	//
	IF _CmdParams[2] = _LiteralString THEN
		// file1.cnc XYZ H +0250.00 +0000.00 +0500.00 +0000.00 +0045.00 +0180.00
		stCommand.StartPos.dX:=STRING_TO_LREAL(_CmdParams[3]);
		stCommand.StartPos.dY:=STRING_TO_LREAL(_CmdParams[4]);
		stCommand.StartPos.dZ:=STRING_TO_LREAL(_CmdParams[5]);
		stCommand.StartPos.dA:=STRING_TO_LREAL(_CmdParams[6]);
		stCommand.StartPos.dB:=STRING_TO_LREAL(_CmdParams[7]);
		stCommand.StartPos.dC:=STRING_TO_LREAL(_CmdParams[8]);
	ELSIF _CmdParams[2] = _VariableString THEN
		// file2.cnc ADD V S 025
		IF _CmdParams[3] = _StoredPositionsString THEN
			//_ArrayType:=DUT_Command_ArrayType.StoredPosition;
			stCommand.StartPos.dX:=PersistentVars.StoredPositions[STRING_TO_INT(_CmdParams[4])].Position.X; // TODO try to remove this reference to global vars
			stCommand.StartPos.dY:=PersistentVars.StoredPositions[STRING_TO_INT(_CmdParams[4])].Position.Y;
			stCommand.StartPos.dZ:=PersistentVars.StoredPositions[STRING_TO_INT(_CmdParams[4])].Position.Z;
			stCommand.StartPos.dA:=PersistentVars.StoredPositions[STRING_TO_INT(_CmdParams[4])].Position.A;
			stCommand.StartPos.dB:=PersistentVars.StoredPositions[STRING_TO_INT(_CmdParams[4])].Position.B;
			stCommand.StartPos.dC:=PersistentVars.StoredPositions[STRING_TO_INT(_CmdParams[4])].Position.C;
		ELSIF _CmdParams[3] = _VisionRegistersString THEN
			//_ArrayType:=DUT_Command_ArrayType.Vision;
			stCommand.StartPos.dX:=PersistentVars.VisionRegisters[STRING_TO_INT(_CmdParams[4])].Position.X;
			stCommand.StartPos.dY:=PersistentVars.VisionRegisters[STRING_TO_INT(_CmdParams[4])].Position.Y;
			stCommand.StartPos.dZ:=PersistentVars.VisionRegisters[STRING_TO_INT(_CmdParams[4])].Position.Z;
			stCommand.StartPos.dA:=PersistentVars.VisionRegisters[STRING_TO_INT(_CmdParams[4])].Position.A;
			stCommand.StartPos.dB:=PersistentVars.VisionRegisters[STRING_TO_INT(_CmdParams[4])].Position.B;
			stCommand.StartPos.dC:=PersistentVars.VisionRegisters[STRING_TO_INT(_CmdParams[4])].Position.C;
		ELSIF _CmdParams[3] = _FlagsString THEN
			//_ArrayType:=DUT_Command_ArrayType.Flag;
		ELSE
			Error := TRUE;
			ErrorDescription:='No array type provided';
		END_IF
	ELSE
		Error := TRUE;
		ErrorDescription:='No variable type provided';
	END_IF
	
ELSE
	Error := TRUE;
	ErrorDescription:='Command string format incorrect';
	
END_IF
                  
END_FUNCTION_BLOCK

FUNCTION F_SplitCmd : ARRAY [0..GVL.COMMAND_LEN] OF STRING
VAR_INPUT
    Command: STRING(GVL.COMMAND_LEN);
	Delimiter: STRING(1):=' ';
END_VAR
VAR
	_Command: STRING(GVL.COMMAND_LEN);
	_DelimPos: INT;
	_i, _j, _k: INT;
END_VAR
VAR CONSTANT
	_SpaceChar: STRING(1):=' ';
END_VAR

                    // grab a copy
// TODO do we need to do this? cant we just operate on the input?
_Command := Command;

// ex. 123 456 789 0 123 456 879 0
WHILE LEN(_Command) > 0  AND _i < GVL.COMMAND_LEN DO
	// find the delimiter
	_DelimPos := FIND(_Command, Delimiter);
	// don't copy empty commands
	IF _DelimPos > 1 THEN
		// copy the command into the array position
		F_SplitCmd[_i] := MID(STR:=_Command, LEN:=_DelimPos - 1, POS:=1);
		// trim the command off the front of the string
		_Command := DELETE(STR:=_Command, LEN:=_DelimPos, POS:=1);
		// increment the index and get ready for the next
		_i := _i + 1;
	ELSIF _DelimPos = 1 OR FIND(_Command, _SpaceChar) = 1 THEN
		// don't do anything with a stray delimiter or a space at the  start of the next command
		// trim the command off the space at the front of the string
		_Command := DELETE(STR:=_Command, LEN:=LEN(_SpaceChar), POS:=1);
	ELSIF _DelimPos = 0 AND LEN(_Command) > 0 THEN
		// copy the last command into the array position and return
		F_SplitCmd[_i] := MID(STR:=_Command, LEN:=LEN(_Command), POS:=1);
		// trim the command off the front of the string
		_Command := DELETE(STR:=_Command, LEN:=_DelimPos, POS:=1);
		// increment the index and get ready for the next
		_i := _i + 1;
		RETURN;
	ELSE
		RETURN;
	END_IF
END_WHILE
                  
END_FUNCTION

FUNCTION BuildVarSetCmd : STRING(GVL.COMMAND_LEN)
VAR_INPUT
	stCommand: ST_VarSetCmd;
END_VAR
VAR
    _Command: STRING(GVL.COMMAND_LEN);
END_VAR
VAR CONSTANT
	_Delimiter: STRING:=' ';
	_ArrayTypeS: STRING(3):='STO';
	_ArrayTypeV: STRING(3):='VIS';
	_ArrayTypeF: STRING(3):='FLG';
END_VAR

                    // S|V|F index x y z a b c
// S 0000 +0000.00 +0000.00 +0000.00 +0000.00 +0000.00 +0000.00 
// V 0000 +0000.00 +0000.00 +0000.00 +0000.00 +0000.00 +0000.00 
// F 0000 1

// clear the command
_Command:='';

// build the command
CASE stCommand.ArrayType OF
	DUT_Command_ArrayType.StoredPosition:
		F_AddElement(_Command, _Delimiter, _ArrayTypeS);
	DUT_Command_ArrayType.VisionRegister:
		F_AddElement(_Command, _Delimiter, _ArrayTypeV);
	DUT_Command_ArrayType.Flag:
		F_AddElement(_Command, _Delimiter, _ArrayTypeF);
END_CASE

// add the array index
F_AddElement(_Command, _Delimiter, INT_TO_STRING(stCommand.ArrayIndex));

// add the coordinates
IF stCommand.ArrayType = DUT_Command_ArrayType.StoredPosition 
	OR stCommand.ArrayType = DUT_Command_ArrayType.VisionRegister THEN
		F_AddElement(_Command, _Delimiter, LREAL_TO_STRING(stCommand.Coordinates.X));
		F_AddElement(_Command, _Delimiter, LREAL_TO_STRING(stCommand.Coordinates.Y));
		F_AddElement(_Command, _Delimiter, LREAL_TO_STRING(stCommand.Coordinates.Z));
		F_AddElement(_Command, _Delimiter, LREAL_TO_STRING(stCommand.Coordinates.A));
		F_AddElement(_Command, _Delimiter, LREAL_TO_STRING(stCommand.Coordinates.B));
		F_AddElement(_Command, _Delimiter, LREAL_TO_STRING(stCommand.Coordinates.C));
		
ELSIF stCommand.ArrayType = DUT_Command_ArrayType.Flag THEN
		// we only send the x for readability. it will work if we send them all.
		F_AddElement(_Command, _Delimiter, LREAL_TO_STRING(stCommand.Coordinates.X));
		
END_IF

// set function equal to command
BuildVarSetCmd := _Command;
                  
END_FUNCTION

FUNCTION_BLOCK LogicCmdProcessor EXTENDS Module
VAR_IN_OUT
	CmdProcessor: CommandProcessor;
	CmdIO: ST_LogicCmdIO;
END_VAR
VAR_INPUT
	Command: STRING(GVL.COMMAND_LEN):='';
END_VAR
VAR_OUTPUT
END_VAR
VAR
	_UnitModeCurrentState: PACK_ML.State;
	_ParseLogicCmd: ParseLogicCmd;
	_ThenFunctionProcessed: BOOL;
END_VAR
VAR CONSTANT
	_STEP_DONE: 		INT := 1000;
	_STEP_IDLE: 		INT := 0000;
	_STEP_COMMAND: 		INT := 0010;
	_STEP_ERR: 			INT := 0020;
	_STEP_EVAL_IN:		INT := 0100;
	_STEP_EVAL_REG:		INT := 0110;
	_STEP_EVAL_CNT:		INT := 0120;
	_STEP_PROC_THEN:	INT := 0200;
	_STEP_PROC_ELSE:	INT := 0210;
	_STEP_PROC_OUT:		INT := 0300;
	_STEP_PROC_JMP:		INT := 0310;
	_STEP_PROC_CNT:		INT := 0320;
	_STEP_PROC_REG:		INT := 0330;
	_STEP_PROC_NOP:		INT := 0340;
END_VAR

                    SUPER^();

// PackML state machine implementation
_UnitModeCurrentState := SUPER^._UnitMode.CurrentState;

//
CASE SUPER^._SeqMain OF
	
    _STEP_DONE:
		SUPER^._SeqMain := _STEP_IDLE;
        
    _STEP_IDLE:
		// wait here until commanded to start
        
    _STEP_COMMAND:
		_ParseLogicCmd(Command:=Command);
		
		CASE _ParseLogicCmd.stCommand.IF_Condition OF
			E_LogicIfCondition.PASS:
				SUPER^._SeqMain := _STEP_PROC_THEN;
			E_LogicIfCondition.INPUT:
				SUPER^._SeqMain := _STEP_EVAL_IN;
			E_LogicIfCondition.REGISTER:
				SUPER^._SeqMain := _STEP_EVAL_REG;
			E_LogicIfCondition.COUNTER:
				SUPER^._SeqMain := _STEP_EVAL_CNT;
		END_CASE
		
		//
		_ThenFunctionProcessed := FALSE;
		
	_STEP_EVAL_IN:
		CASE _ParseLogicCmd.stCommand.IF_Condition_Operator OF
			E_LogicIfConditionOperator.EQU:
				IF CmdIO.Input[_ParseLogicCmd.stCommand.IF_Condition_Idx] 
					= UDINT_TO_BOOL(_ParseLogicCmd.stCommand.IF_Condition_Operator_Value) THEN
						SUPER^._SeqMain := _STEP_PROC_THEN;
				ELSE
					SUPER^._SeqMain := _STEP_PROC_ELSE;
				END_IF
			E_LogicIfConditionOperator.GRE:
				IF CmdIO.Input[_ParseLogicCmd.stCommand.IF_Condition_Idx] 
					>= UDINT_TO_BOOL(_ParseLogicCmd.stCommand.IF_Condition_Operator_Value) THEN
						SUPER^._SeqMain := _STEP_PROC_THEN;
				ELSE
					SUPER^._SeqMain := _STEP_PROC_ELSE;
				END_IF
			E_LogicIfConditionOperator.GRT:
				IF CmdIO.Input[_ParseLogicCmd.stCommand.IF_Condition_Idx] 
					> UDINT_TO_BOOL(_ParseLogicCmd.stCommand.IF_Condition_Operator_Value) THEN
						SUPER^._SeqMain := _STEP_PROC_THEN;
				ELSE
					SUPER^._SeqMain := _STEP_PROC_ELSE;
				END_IF
			E_LogicIfConditionOperator.LEQ:
				IF CmdIO.Input[_ParseLogicCmd.stCommand.IF_Condition_Idx] 
					<= UDINT_TO_BOOL(_ParseLogicCmd.stCommand.IF_Condition_Operator_Value) THEN
						SUPER^._SeqMain := _STEP_PROC_THEN;
				ELSE
					SUPER^._SeqMain := _STEP_PROC_ELSE;
				END_IF
			E_LogicIfConditionOperator.LES:
				IF CmdIO.Input[_ParseLogicCmd.stCommand.IF_Condition_Idx] 
					< UDINT_TO_BOOL(_ParseLogicCmd.stCommand.IF_Condition_Operator_Value) THEN
						SUPER^._SeqMain := _STEP_PROC_THEN;
				ELSE
					SUPER^._SeqMain := _STEP_PROC_ELSE;
				END_IF
		END_CASE
		
	_STEP_EVAL_REG:
		CASE _ParseLogicCmd.stCommand.IF_Condition_Operator OF
			E_LogicIfConditionOperator.EQU:
				IF CmdIO.Register[_ParseLogicCmd.stCommand.IF_Condition_Idx] 
					= _ParseLogicCmd.stCommand.IF_Condition_Operator_Value THEN
						SUPER^._SeqMain := _STEP_PROC_THEN;
				ELSE
					SUPER^._SeqMain := _STEP_PROC_ELSE;
				END_IF
			E_LogicIfConditionOperator.GRE:
				IF CmdIO.Register[_ParseLogicCmd.stCommand.IF_Condition_Idx] 
					>= _ParseLogicCmd.stCommand.IF_Condition_Operator_Value THEN
						SUPER^._SeqMain := _STEP_PROC_THEN;
				ELSE
					SUPER^._SeqMain := _STEP_PROC_ELSE;
				END_IF
			E_LogicIfConditionOperator.GRT:
				IF CmdIO.Register[_ParseLogicCmd.stCommand.IF_Condition_Idx] 
					> _ParseLogicCmd.stCommand.IF_Condition_Operator_Value THEN
						SUPER^._SeqMain := _STEP_PROC_THEN;
				ELSE
					SUPER^._SeqMain := _STEP_PROC_ELSE;
				END_IF
			E_LogicIfConditionOperator.LEQ:
				IF CmdIO.Register[_ParseLogicCmd.stCommand.IF_Condition_Idx] 
					<= _ParseLogicCmd.stCommand.IF_Condition_Operator_Value THEN
						SUPER^._SeqMain := _STEP_PROC_THEN;
				ELSE
					SUPER^._SeqMain := _STEP_PROC_ELSE;
				END_IF
			E_LogicIfConditionOperator.LES:
				IF CmdIO.Register[_ParseLogicCmd.stCommand.IF_Condition_Idx] 
					< _ParseLogicCmd.stCommand.IF_Condition_Operator_Value THEN
						SUPER^._SeqMain := _STEP_PROC_THEN;
				ELSE
					SUPER^._SeqMain := _STEP_PROC_ELSE;
				END_IF
		END_CASE
		
	_STEP_EVAL_CNT:
		CASE _ParseLogicCmd.stCommand.IF_Condition_Operator OF
			E_LogicIfConditionOperator.EQU:
				IF CmdIO.Counter[_ParseLogicCmd.stCommand.IF_Condition_Idx] 
					= _ParseLogicCmd.stCommand.IF_Condition_Operator_Value THEN
						SUPER^._SeqMain := _STEP_PROC_THEN;
				ELSE
					SUPER^._SeqMain := _STEP_PROC_ELSE;
				END_IF
			E_LogicIfConditionOperator.GRE:
				IF CmdIO.Counter[_ParseLogicCmd.stCommand.IF_Condition_Idx] 
					>= _ParseLogicCmd.stCommand.IF_Condition_Operator_Value THEN
						SUPER^._SeqMain := _STEP_PROC_THEN;
				ELSE
					SUPER^._SeqMain := _STEP_PROC_ELSE;
				END_IF
			E_LogicIfConditionOperator.GRT:
				IF CmdIO.Counter[_ParseLogicCmd.stCommand.IF_Condition_Idx] 
					> _ParseLogicCmd.stCommand.IF_Condition_Operator_Value THEN
						SUPER^._SeqMain := _STEP_PROC_THEN;
				ELSE
					SUPER^._SeqMain := _STEP_PROC_ELSE;
				END_IF
			E_LogicIfConditionOperator.LEQ:
				IF CmdIO.Counter[_ParseLogicCmd.stCommand.IF_Condition_Idx] 
					<= _ParseLogicCmd.stCommand.IF_Condition_Operator_Value THEN
						SUPER^._SeqMain := _STEP_PROC_THEN;
				ELSE
					SUPER^._SeqMain := _STEP_PROC_ELSE;
				END_IF
			E_LogicIfConditionOperator.LES:
				IF CmdIO.Counter[_ParseLogicCmd.stCommand.IF_Condition_Idx] 
					< _ParseLogicCmd.stCommand.IF_Condition_Operator_Value THEN
						SUPER^._SeqMain := _STEP_PROC_THEN;
				ELSE
					SUPER^._SeqMain := _STEP_PROC_ELSE;
				END_IF
		END_CASE
		
	_STEP_PROC_THEN:
		//
		_ThenFunctionProcessed := TRUE;
		//
		CASE _ParseLogicCmd.stCommand.THEN_Function OF
			E_LogicFunction.OUTPUT:
				SUPER^._SeqMain := _STEP_PROC_OUT;
			E_LogicFunction.REGISTER:
				SUPER^._SeqMain := _STEP_PROC_REG;
			E_LogicFunction.CNTUP:
				SUPER^._SeqMain := _STEP_PROC_CNT;
			E_LogicFunction.CNTDN:
				SUPER^._SeqMain := _STEP_PROC_CNT;
			E_LogicFunction.CNTRST:
				SUPER^._SeqMain := _STEP_PROC_CNT;
			E_LogicFunction.JUMP:
				SUPER^._SeqMain := _STEP_PROC_JMP;
			E_LogicFunction.NOP:
				SUPER^._SeqMain := _STEP_PROC_NOP;
		END_CASE;
				
	_STEP_PROC_ELSE:
		CASE _ParseLogicCmd.stCommand.ELSE_Function OF
			E_LogicFunction.OUTPUT:
				SUPER^._SeqMain := _STEP_PROC_OUT;
			E_LogicFunction.REGISTER:
				SUPER^._SeqMain := _STEP_PROC_REG;
			E_LogicFunction.CNTUP:
				SUPER^._SeqMain := _STEP_PROC_CNT;
			E_LogicFunction.CNTDN:
				SUPER^._SeqMain := _STEP_PROC_CNT;
			E_LogicFunction.CNTRST:
				SUPER^._SeqMain := _STEP_PROC_CNT;
			E_LogicFunction.JUMP:
				SUPER^._SeqMain := _STEP_PROC_JMP;
			E_LogicFunction.NOP:
				SUPER^._SeqMain := _STEP_PROC_NOP;
		END_CASE;
		
	_STEP_PROC_OUT:
		IF _ThenFunctionProcessed THEN
			CmdIO.Output[_ParseLogicCmd.stCommand.THEN_Function_Idx] 
				:= UDINT_TO_BOOL(_ParseLogicCmd.stCommand.THEN_Function_Value);
		ELSE
			CmdIO.Output[_ParseLogicCmd.stCommand.ELSE_Function_Idx] 
				:= UDINT_TO_BOOL(_ParseLogicCmd.stCommand.ELSE_Function_Value);
		END_IF
		// next, please
		SUPER^._SeqMain := _STEP_DONE;
		
	_STEP_PROC_REG:
		IF _ThenFunctionProcessed THEN
			CmdIO.Register[_ParseLogicCmd.stCommand.THEN_Function_Idx] 
				:= _ParseLogicCmd.stCommand.THEN_Function_Value;
		ELSE
			CmdIO.Register[_ParseLogicCmd.stCommand.ELSE_Function_Idx] 
				:= _ParseLogicCmd.stCommand.ELSE_Function_Value;
		END_IF
		// next, please
		SUPER^._SeqMain := _STEP_DONE;
		
	_STEP_PROC_CNT:	
		IF _ThenFunctionProcessed THEN
			CASE _ParseLogicCmd.stCommand.THEN_Function OF
				E_LogicFunction.CNTUP:
					CmdIO.Counter[_ParseLogicCmd.stCommand.THEN_Function_Idx] 
						:= CmdIO.Counter[_ParseLogicCmd.stCommand.THEN_Function_Idx] + 1;
				E_LogicFunction.CNTDN:
					CmdIO.Counter[_ParseLogicCmd.stCommand.THEN_Function_Idx] 
						:= CmdIO.Counter[_ParseLogicCmd.stCommand.THEN_Function_Idx] - 1;
				E_LogicFunction.CNTRST:
					CmdIO.Counter[_ParseLogicCmd.stCommand.THEN_Function_Idx] 
						:= 0;
			END_CASE
		ELSE
			CASE _ParseLogicCmd.stCommand.ELSE_Function OF
				E_LogicFunction.CNTUP:
					CmdIO.Counter[_ParseLogicCmd.stCommand.ELSE_Function_Idx] 
						:= CmdIO.Counter[_ParseLogicCmd.stCommand.ELSE_Function_Idx] + 1;
				E_LogicFunction.CNTDN:
					CmdIO.Counter[_ParseLogicCmd.stCommand.ELSE_Function_Idx] 
						:= CmdIO.Counter[_ParseLogicCmd.stCommand.ELSE_Function_Idx] - 1;
				E_LogicFunction.CNTRST:
					CmdIO.Counter[_ParseLogicCmd.stCommand.ELSE_Function_Idx] 
						:= 0;
			END_CASE
		END_IF
		// next, please
		SUPER^._SeqMain := _STEP_DONE;
		
	_STEP_PROC_JMP:
		// TODO need to create a function in the command processor to change the next step
		// leaving this guy dead for now.
		IF _ThenFunctionProcessed THEN
			CmdProcessor.M_SetNextCommand(CommandNumber:=INT_TO_UINT(_ParseLogicCmd.stCommand.THEN_Function_Idx));
		ELSE
			CmdProcessor.M_SetNextCommand(CommandNumber:=INT_TO_UINT(_ParseLogicCmd.stCommand.ELSE_Function_Idx));
		END_IF
		// next, please
		SUPER^._SeqMain := _STEP_DONE;
		
	_STEP_PROC_NOP:
		IF _ThenFunctionProcessed THEN
			//
		ELSE
			//
		END_IF
		// next, please
		SUPER^._SeqMain := _STEP_DONE;

END_CASE
                  

METHOD PROTECTED M_SetPackML : BOOL
                          SUPER^._UnitMode(	sName := 'Logic Processor',
				eInitialState := PACK_ML.State.Idle,
				xActive := TRUE);
                        
END_METHOD

METHOD PROTECTED M_Complete : BOOL
                          // once complete, reset to get back to idle
SUPER^._UnitMode.Reset();
                        
END_METHOD

METHOD PROTECTED M_Execute : BOOL
                          // here we want to execute our commands/jobs/etc and set completed when done.
IF SUPER^._SeqMain =_STEP_IDLE THEN
	SUPER^.M_StateComplete();
END_IF
                        
END_METHOD

METHOD PROTECTED M_Starting : BOOL
                          // here we want to clear things and get ready for the execute state
// I can consider this the "INIT" state
SUPER^._SeqMain := _STEP_COMMAND;
SUPER^.M_StateComplete();
                        
END_METHOD
END_FUNCTION_BLOCK

FUNCTION F_AddElement
VAR_IN_OUT
	Command: STRING(GVL.COMMAND_LEN);
END_VAR
VAR_INPUT
	Delimiter: STRING(1):=' '; // default to space
	Element: STRING(GVL.COMMAND_LEN);
END_VAR
VAR
END_VAR

                    //
// input
// 	Element: 'bar'
// 	Delimiter: ','
// 	Command: 'foo'
//
// output
// 	Command: 'foo,bar'
//

Command:=CONCAT(Command, Element);
Command:=CONCAT(Command, Delimiter);
                  
END_FUNCTION

FUNCTION BuildMoveCmd : STRING(GVL.COMMAND_LEN);
VAR_INPUT
	stCommand: ST_MoveCmd;
END_VAR
VAR
	_Command : STRING(GVL.COMMAND_LEN);
END_VAR
VAR CONSTANT
	_Delimiter: STRING:=' ';
	_MoveTypeD: STRING(3):='DIR';
	_MoveTypeL: STRING(3):='LIN';
	_MoveTypeC: STRING(3):='CIR';
	_ChangeTypeA: STRING(3):='ABS';
	_ChangeTypeR: STRING(3):='REL';
	_CoordSystemAcs: STRING(3):='ACS';
	_CoordSystemMcs: STRING(3):='MCS';
	_CoordSystemPc1: STRING(3):='PC1';
	_CoordSystemPc2: STRING(3):='PC2';
	_CoordSystemTcs: STRING(3):='TCS';
	_CoordSystemWcs: STRING(3):='WCS';
	_CoordSystemIcs: STRING(3):='ICS';
	_CoordTypeH: STRING(3):='LIT';
	_CoordTypeV: STRING(3):='VAR';
	_ArrayTypeS: STRING(3):='STO';
	_ArrayTypeV: STRING(3):='VIS';
	_ArrayTypeF: STRING(3):='FLG';
	_CircleModeBor: STRING(3):='BOR';
	_CircleModeCen: STRING(3):='CEN';
	_CircleModeRad: STRING(3):='RAD';
	_PathChoiceClw: STRING(3):='CLW';
	_PathChoiceCcw: STRING(3):='CCW';
END_VAR

                    // D is direct move. L is linear move. C is a circular move
// R is relative position. A is absolute position
// V is variable coordinated. H is a hardcoded coordinated
// S is stored position array. V is vision register array.
// D|L|C R|A Speed CoordSystem X0000.00 Y0000.00 Z0000.00 A0000.00 B0000.00 C0000.00 BOR|CEN|RAD CCW|CLW X0000.00 Y0000.00 Z0000.00 A0000.00 B0000.00 C0000.00
// 'D A 010 MCS H +0250.00 +0000.00 +0500.00 +0000.00 +0045.00 +0180.00'
// 'C R 010 MCS H +0250.00 +0000.00 +0500.00 +0000.00 +0045.00 +0180.00 BOR CLW H +0250.00 +0000.00 +0500.00 +0000.00 +0045.00 +0180.00'
// 'D A 010 MCS V S 025'
// 'D A 010 MCS V V 033'
// 'C R 010 MCS V S 002 BOR CLW V S 005'
// 'C R 010 MCS V S 003 BOR CLW V V 006'
// 'C R 010 MCS V S 015 BOR CLW H +0250.00 +0000.00 +0500.00 +0000.00 +0045.00 +0180.00'
// 'C R 010 MCS H +0250.00 +0000.00 +0500.00 +0000.00 +0045.00 +0180.00 BOR CLW V V 022'

//
_Command := '';

//
CASE stCommand.MoveType OF
	DUT_Command_MoveType.DirectMove:
		F_AddElement(_Command, _Delimiter, _MoveTypeD);
	DUT_Command_MoveType.LinearMove:
		F_AddElement(_Command, _Delimiter, _MoveTypeL);
	DUT_Command_MoveType.CircularMove:
		F_AddElement(_Command, _Delimiter, _MoveTypeC);
END_CASE

//
CASE stCommand.PositionType OF
	DUT_Command_PositionType.AbsolutePosition:
		F_AddElement(_Command, _Delimiter, _ChangeTypeA);
	DUT_Command_PositionType.RelativePosition:
		F_AddElement(_Command, _Delimiter, _ChangeTypeR);
END_CASE

//
F_AddElement(_Command, _Delimiter, LREAL_TO_STRING(stCommand.Speed));

//
CASE stCommand.CoordSystem OF
	SMC_COORD_SYSTEM.ACS:
		F_AddElement(_Command, _Delimiter, _CoordSystemAcs);
	SMC_COORD_SYSTEM.MCS:
		F_AddElement(_Command, _Delimiter, _CoordSystemMcs);
	SMC_COORD_SYSTEM.PCS_1:
		F_AddElement(_Command, _Delimiter, _CoordSystemPc1);
	SMC_COORD_SYSTEM.PCS_2:
		F_AddElement(_Command, _Delimiter, _CoordSystemPc2);
	SMC_COORD_SYSTEM.TCS:
		F_AddElement(_Command, _Delimiter, _CoordSystemTcs);
	SMC_COORD_SYSTEM.WCS:
		F_AddElement(_Command, _Delimiter, _CoordSystemWcs);
	SMC_COORD_SYSTEM.ICS:
		F_AddElement(_Command, _Delimiter, _CoordSystemIcs);
END_CASE

//
CASE stCommand.CoordinateType OF
	DUT_Command_CoordinateType.Literal:
		F_AddElement(_Command, _Delimiter, _CoordTypeH);
		F_AddElement(_Command, _Delimiter, LREAL_TO_STRING(stCommand.CoordRef.X));
		F_AddElement(_Command, _Delimiter, LREAL_TO_STRING(stCommand.CoordRef.Y));
		F_AddElement(_Command, _Delimiter, LREAL_TO_STRING(stCommand.CoordRef.Z));
		F_AddElement(_Command, _Delimiter, LREAL_TO_STRING(stCommand.CoordRef.A));
		F_AddElement(_Command, _Delimiter, LREAL_TO_STRING(stCommand.CoordRef.B));
		F_AddElement(_Command, _Delimiter, LREAL_TO_STRING(stCommand.CoordRef.C));
		
	DUT_Command_CoordinateType.Variable:
		F_AddElement(_Command, _Delimiter, _CoordTypeV);
		CASE stCommand.ArrayType OF
			DUT_Command_ArrayType.StoredPosition:
				F_AddElement(_Command, _Delimiter, _ArrayTypeS);
			DUT_Command_ArrayType.VisionRegister:
				F_AddElement(_Command, _Delimiter, _ArrayTypeV);
			DUT_Command_ArrayType.Flag:
				// on damn
		END_CASE
		F_AddElement(_Command, _Delimiter, UDINT_TO_STRING(stCommand.ArrayIndex));
		
END_CASE

// only add if move type is circle
IF stCommand.MoveType = DUT_Command_MoveType.CircularMove THEN
	//
	CASE stCommand.CircleMode OF
		SMC_CIRC_MODE.BORDER:
			F_AddElement(_Command, _Delimiter, _CircleModeBor);
		SMC_CIRC_MODE.CENTER:
			F_AddElement(_Command, _Delimiter, _CircleModeCen);
		SMC_CIRC_MODE.RADIUS:
			F_AddElement(_Command, _Delimiter, _CircleModeRad);
	END_CASE
	//
	CASE stCommand.PathChoice OF
		MC_CIRC_PATHCHOICE.CLOCKWISE:
			F_AddElement(_Command, _Delimiter, _PathChoiceClw);
		MC_CIRC_PATHCHOICE.COUNTER_CLOCKWISE:
			F_AddElement(_Command, _Delimiter, _PathChoiceCcw);
	END_CASE
	//
	CASE stCommand.CircularCoordinateType OF
		DUT_Command_CoordinateType.Literal:
			F_AddElement(_Command, _Delimiter, _CoordTypeH);
			F_AddElement(_Command, _Delimiter, LREAL_TO_STRING(stCommand.CoordRef2.X));
			F_AddElement(_Command, _Delimiter, LREAL_TO_STRING(stCommand.CoordRef2.Y));
			F_AddElement(_Command, _Delimiter, LREAL_TO_STRING(stCommand.CoordRef2.Z));
			F_AddElement(_Command, _Delimiter, LREAL_TO_STRING(stCommand.CoordRef2.A));
			F_AddElement(_Command, _Delimiter, LREAL_TO_STRING(stCommand.CoordRef2.B));
			F_AddElement(_Command, _Delimiter, LREAL_TO_STRING(stCommand.CoordRef2.C));
			
		DUT_Command_CoordinateType.Variable:
			F_AddElement(_Command, _Delimiter, _CoordTypeV);
			CASE stCommand.CircularArrayType OF
				DUT_Command_ArrayType.StoredPosition:
					F_AddElement(_Command, _Delimiter, _ArrayTypeS);
				DUT_Command_ArrayType.VisionRegister:
					F_AddElement(_Command, _Delimiter, _ArrayTypeV);
				DUT_Command_ArrayType.Flag:
					// oh damn
			END_CASE
			F_AddElement(_Command, _Delimiter, UDINT_TO_STRING(stCommand.CircularArrayIndex));
			
	END_CASE

END_IF

// set function equal to command
BuildMoveCmd := _Command;
                  
END_FUNCTION

FUNCTION F_RoundLreal : LREAL
VAR_INPUT
   rIn : LREAL;      
   Digit: INT;         
END_VAR

VAR
   d1 : DINT;
   r0,r1,r2,Rdigit: LREAL;               
END_VAR

                    // https://forge.codesys.com/forge/talk/Engineering/thread/8d1ee86294/
rdigit   :=INT_TO_LREAL(Digit);
r0 := EXPT(10,rdigit); 
r1 := rIn * r0;
d1 := TRUNC(r1);
r2 := DINT_TO_LREAL(d1);
F_RoundLreal := r2 / r0;
                  
END_FUNCTION

FUNCTION_BLOCK ParseLogicCmd
VAR_INPUT
	Command: STRING(GVL.COMMAND_LEN);
END_VAR
VAR_OUTPUT
	stCommand: ST_LogicCmd;
	Error: BOOL;
	ErrorDescription: STRING;
END_VAR
VAR
	_CmdParams: ARRAY [0..GVL.COMMAND_LEN] OF STRING;
	_i, _j, _k: INT;
END_VAR

                    // IF PASS|INPUT|REGISTER|COUNTER <index> >|<|=|>=|<= <value>
// THEN OUTPUT|JUMP|CNTUP|CNTDN|CNTRST|REGISTER|NOP <index> <value>
// ELSE OUTPUT|JUMP|CNTUP|CNTDN|CNTRST|REGISTER|NOP <index> <value>
//
// IF_Condition
// IF_Condition_Idx
// IF_Condition_Operator
// IF_Condition_Operator_Compare
// THEN_Function
// THEN_Function_Value
// THEN_Function_Idx
// ELSE_Function
// ELSE_Function_Idx
// ELSE_Function_Value

Error:=FALSE;
ErrorDescription:='';

// split command string into commands
_CmdParams:=F_SplitCmd(Command:=Command);

//
_i := 0;

// disregard the 'IF'
_i := _i + 1;

//
IF _CmdParams[_i] = TO_STRING(E_LogicIfCondition.PASS) THEN
	stCommand.IF_Condition := E_LogicIfCondition.PASS;
ELSIF  _CmdParams[_i] = TO_STRING(E_LogicIfCondition.INPUT) THEN
	stCommand.IF_Condition := E_LogicIfCondition.INPUT;
ELSIF  _CmdParams[_i] = TO_STRING(E_LogicIfCondition.REGISTER) THEN
	stCommand.IF_Condition := E_LogicIfCondition.REGISTER;
ELSIF  _CmdParams[_i] = TO_STRING(E_LogicIfCondition.COUNTER) THEN
	stCommand.IF_Condition := E_LogicIfCondition.COUNTER;
END_IF
_i := _i + 1;

//
IF stCommand.IF_Condition <> E_LogicIfCondition.PASS THEN
	
	//
	stCommand.IF_Condition_Idx := STRING_TO_INT(_CmdParams[_i]);
	_i := _i + 1;
	
	//
	IF _CmdParams[_i] = TO_STRING(E_LogicIfConditionOperator.GRT) THEN
		stCommand.IF_Condition_Operator := E_LogicIfConditionOperator.GRT;
	ELSIF _CmdParams[_i] = TO_STRING(E_LogicIfConditionOperator.LES) THEN
		stCommand.IF_Condition_Operator := E_LogicIfConditionOperator.LES;                   
	ELSIF _CmdParams[_i] = TO_STRING(E_LogicIfConditionOperator.EQU) THEN
		stCommand.IF_Condition_Operator := E_LogicIfConditionOperator.EQU;
	ELSIF _CmdParams[_i] = TO_STRING(E_LogicIfConditionOperator.GRE) THEN
		stCommand.IF_Condition_Operator := E_LogicIfConditionOperator.GRE;
	ELSIF _CmdParams[_i] = TO_STRING(E_LogicIfConditionOperator.LEQ) THEN
		stCommand.IF_Condition_Operator := E_LogicIfConditionOperator.LEQ;
	END_IF
	_i := _i + 1;
	
	//
	stCommand.IF_Condition_Operator_Value := STRING_TO_UDINT(_CmdParams[_i]);
	_i := _i + 1;
	
END_IF

// disregard the 'THEN'
_i := _i + 1;

//
IF _CmdParams[_i] = TO_STRING(E_LogicFunction.OUTPUT) THEN
	stCommand.THEN_Function := E_LogicFunction.OUTPUT;
ELSIF _CmdParams[_i] = TO_STRING(E_LogicFunction.JUMP) THEN
	stCommand.THEN_Function := E_LogicFunction.JUMP;                 
ELSIF _CmdParams[_i] = TO_STRING(E_LogicFunction.CNTUP) THEN
	stCommand.THEN_Function := E_LogicFunction.CNTUP;
ELSIF _CmdParams[_i] = TO_STRING(E_LogicFunction.CNTDN) THEN
	stCommand.THEN_Function := E_LogicFunction.CNTDN;
ELSIF _CmdParams[_i] = TO_STRING(E_LogicFunction.CNTRST) THEN
	stCommand.THEN_Function := E_LogicFunction.CNTRST;
ELSIF _CmdParams[_i] = TO_STRING(E_LogicFunction.REGISTER) THEN
	stCommand.THEN_Function := E_LogicFunction.REGISTER;
ELSIF _CmdParams[_i] = TO_STRING(E_LogicFunction.NOP) THEN
	stCommand.THEN_Function := E_LogicFunction.NOP;
END_IF
_i := _i + 1;

//
IF stCommand.THEN_Function <> E_LogicFunction.NOP THEN
	stCommand.THEN_Function_Idx := STRING_TO_INT(_CmdParams[_i]);
	_i := _i + 1;
	IF stCommand.THEN_Function = E_LogicFunction.OUTPUT 
		OR stCommand.THEN_Function = E_LogicFunction.REGISTER THEN
			stCommand.THEN_Function_Value := STRING_TO_UDINT(_CmdParams[_i]);
			_i := _i + 1;
	END_IF
END_IF

// disregard the 'ELSE'
_i := _i + 1;

//
IF _CmdParams[_i] = TO_STRING(E_LogicFunction.OUTPUT) THEN
	stCommand.ELSE_Function := E_LogicFunction.OUTPUT;
ELSIF _CmdParams[_i] = TO_STRING(E_LogicFunction.JUMP) THEN
	stCommand.ELSE_Function := E_LogicFunction.JUMP;                 
ELSIF _CmdParams[_i] = TO_STRING(E_LogicFunction.CNTUP) THEN
	stCommand.ELSE_Function := E_LogicFunction.CNTUP;
ELSIF _CmdParams[_i] = TO_STRING(E_LogicFunction.CNTDN) THEN
	stCommand.ELSE_Function := E_LogicFunction.CNTDN;
ELSIF _CmdParams[_i] = TO_STRING(E_LogicFunction.CNTRST) THEN
	stCommand.ELSE_Function := E_LogicFunction.CNTRST;
ELSIF _CmdParams[_i] = TO_STRING(E_LogicFunction.REGISTER) THEN
	stCommand.ELSE_Function := E_LogicFunction.REGISTER;
ELSIF _CmdParams[_i] = TO_STRING(E_LogicFunction.NOP) THEN
	stCommand.ELSE_Function := E_LogicFunction.NOP;
END_IF
_i := _i + 1;

//
IF stCommand.ELSE_Function <> E_LogicFunction.NOP THEN
	stCommand.ELSE_Function_Idx := STRING_TO_INT(_CmdParams[_i]);
	_i := _i + 1;
	IF stCommand.ELSE_Function = E_LogicFunction.OUTPUT 
		OR stCommand.ELSE_Function = E_LogicFunction.REGISTER THEN
			stCommand.ELSE_Function_Value := STRING_TO_UDINT(_CmdParams[_i]);
			_i := _i + 1;
	END_IF
END_IF
                  
END_FUNCTION_BLOCK

FUNCTION BuildLogicCmd : STRING(GVL.COMMAND_LEN)
VAR_INPUT
	stCommand: ST_LogicCmd;
END_VAR
VAR
    _Command: STRING(GVL.COMMAND_LEN);
END_VAR
VAR CONSTANT
	_Delimiter: STRING:=' ';
END_VAR

                    // IF PASS|INPUT|REGISTER|COUNTER <index> >|<|=|>=|<= <value>
// THEN OUTPUT|JUMP|CNTUP|CNTDN|CNTRST|REGISTER|NOP <index> <value>
// ELSE OUTPUT|JUMP|CNTUP|CNTDN|CNTRST|REGISTER|NOP <index> <value>
//
// IF_Condition
// IF_Condition_Idx
// IF_Condition_Operator
// IF_Condition_Operator_Compare
// THEN_Function
// THEN_Function_Value
// THEN_Function_Idx
// ELSE_Function
// ELSE_Function_Idx
// ELSE_Function_Value

// clear the command
_Command:='';

// build command
F_AddElement(_Command, _Delimiter, 'IF');
F_AddElement(_Command, _Delimiter, TO_STRING(stCommand.IF_Condition));
IF stCommand.IF_Condition <> E_LogicIfCondition.PASS THEN
	F_AddElement(_Command, _Delimiter, INT_TO_STRING(stCommand.IF_Condition_Idx));
	F_AddElement(_Command, _Delimiter, TO_STRING(stCommand.IF_Condition_Operator));
	F_AddElement(_Command, _Delimiter, UDINT_TO_STRING(stCommand.IF_Condition_Operator_Value));
END_IF
F_AddElement(_Command, _Delimiter, 'THEN');
F_AddElement(_Command, _Delimiter, TO_STRING(stCommand.THEN_Function));
IF stCommand.THEN_Function <> E_LogicFunction.NOP THEN
	F_AddElement(_Command, _Delimiter, INT_TO_STRING(stCommand.THEN_Function_Idx));
	IF stCommand.THEN_Function = E_LogicFunction.OUTPUT OR 
		stCommand.THEN_Function = E_LogicFunction.REGISTER THEN
			F_AddElement(_Command, _Delimiter, UDINT_TO_STRING(stCommand.THEN_Function_Value));
	END_IF
END_IF
F_AddElement(_Command, _Delimiter, 'ELSE');
F_AddElement(_Command, _Delimiter, TO_STRING(stCommand.ELSE_Function));
IF stCommand.ELSE_Function <> E_LogicFunction.NOP THEN
	F_AddElement(_Command, _Delimiter, INT_TO_STRING(stCommand.ELSE_Function_Idx));
	IF stCommand.ELSE_Function = E_LogicFunction.OUTPUT 
		OR stCommand.ELSE_Function = E_LogicFunction.REGISTER THEN
			F_AddElement(_Command, _Delimiter, UDINT_TO_STRING(stCommand.ELSE_Function_Value));
	END_IF
END_IF

// set function equal to command
BuildLogicCmd := _Command;
                  
END_FUNCTION

CONFIGURATION Device
  RESOURCE Application ON PLC
(* global variable list GVL *)
{attribute 'qualified_only'}

VAR_GLOBAL CONSTANT
	
	// task scan times
	dwMainInterval: DWORD:=3000; // us TODO reference this in task settings
	dwMotionInterval: DWORD:=50; // us TODO reference this in task settings
	dwVisionInterval: DWORD:=20000; // us TODO reference this in task settings
	dwVisuInterval: DWORD:=100000; // us TODO reference this in task settings
	
	// array sizes
	DIG_OUT_ARR_BEG: INT:=0;
	DIG_OUT_ARR_END: INT:=7;
	DIG_IN_ARR_BEG: INT:=0;
	DIG_IN_ARR_END: INT:=7;
	PROG_CMDS_ARR_BEG: INT:=0;
	PROG_CMDS_ARR_END: INT:=49; // total number of commands in a program
	PROG_ARR_BEG: INT:=0;
	PROG_ARR_END: INT:=19; // total number of programs 
	POS_ARR_BEG: INT:=0;
	POS_ARR_END: INT:=49; // total number of stored positions
	VIS_ARR_BEG: INT:=0;
	VIS_ARR_END: INT:=49; // total number of vision registers
	FLG_ARR_BEG: INT:=0;
	FLG_ARR_END: INT:=49; // total number of flags
	REG_ARR_BEG: INT:=0;
	REG_ARR_END: INT:=49; // total number of registers
	
END_VAR

VAR_GLOBAL CONSTANT
	
	// length of command strings for command processor.
	// if this is reduced then commands may stop working.
	COMMAND_LEN: UINT:=255;

	// stored positions
	POSE_1_IDX: INT:=34; // coordinates of pose 1
	POSE_2_IDX: INT:=35; // coordinates of pose 2
	POSE_3_IDX: INT:=36; // coordinates of pose 3
	POSE_4_IDX: INT:=37; // coordinates of pose 4
	POSE_5_IDX: INT:=38; // coordinates of pose 5
	//RESERVED: INT:=39; // RESERVED
	//RESERVED: INT:=40; // RESERVED
	//RESERVED: INT:=41; // RESERVED
	//RESERVED: INT:=42; // RESERVED
	//RESERVED: INT:=43; // RESERVED
	HOM_POS_IDX: INT:=44; // homing offsets
	DEC_START_POS: INT:=45; // start position for the nc decoder
	TCP_POS_IDX: INT:=46; // tool center point offset
	PC2_POS_IDX: INT:=47; // part 2 coordinate system offset
	PC1_POS_IDX: INT:=48; // part 1 coordinate system offset
	MCS_POS_IDX: INT:=49; // machine (robot) coordinate system offset
	
	// vision registers
	//RESERVED: INT:=VIS_ARR_END-4; // RESERVED
	//RESERVED: INT:=VIS_ARR_END-3; // RESERVED
	//RESERVED: INT:=VIS_ARR_END-2; // RESERVED
	//RESERVED: INT:=VIS_ARR_END-1; // RESERVED
	//RESERVED: INT:=VIS_ARR_END; // RESERVED
	
	// flags
	HOM_TO_POSE_IDX: INT:=44;
	//RESERVED: INT:=45;
	//RESERVED: INT:=46;
	//RESERVED: INT:=47;
	HOME_COMPLETE: INT:=48;
	INIT_POS_IDX: INT:=49;
	
END_VAR

VAR_GLOBAL
	
	//
	PowerOn:BOOL;
	Homing: BOOL;
	Reset: BOOL;
	
	// command IO
	DigitalInput: ARRAY [DIG_IN_ARR_BEG..DIG_IN_ARR_END] OF BOOL;
	DigitalOutput: ARRAY [DIG_OUT_ARR_BEG..DIG_OUT_ARR_END] OF BOOL;
	CmdIO: ST_LogicCmdIO;
	
	// cnc (testing)
	g_x: REAL:=50; // feed rate
	g_y: REAL:=50;
	g_gripper: INT:=0;
	Servo0Position: BYTE;
	
	//
	MoveToPose1: BOOL;
	MoveToPose2: BOOL;
	Pose1: STRING(GVL.COMMAND_LEN);
	Pose2: STRING(GVL.COMMAND_LEN);
	
END_VAR
(* global variable list PersistentVars *)
{attribute 'qualified_only'}
VAR_GLOBAL PERSISTENT RETAIN
	Programs: ARRAY [GVL.PROG_ARR_BEG..GVL.PROG_ARR_END] OF DUT_Program;
	StoredPositions: ARRAY [GVL.POS_ARR_BEG..GVL.POS_ARR_END] OF DUT_StoredPosition;
	VisionRegisters: ARRAY[GVL.VIS_ARR_BEG..GVL.VIS_ARR_END] OF DUT_VisionRegister;
	Flags: ARRAY[GVL.FLG_ARR_BEG..GVL.FLG_ARR_END] OF DUT_Flags;
END_VAR
    TASK MainTask(INTERVAL := T#3ms, PRIORITY := 1);
    TASK SoftMotion_PlanningTask(INTERVAL := T#0.05ms, PRIORITY := 15);
    TASK VISU_TASK(INTERVAL := T#100ms, PRIORITY := 31);
    TASK VisionTask(INTERVAL := T#20ms, PRIORITY := 10);
    PROGRAM _00_Main WITH MainTask : _00_Main;
    PROGRAM _20_Io WITH MainTask : _20_Io;
    PROGRAM _10_Drives WITH SoftMotion_PlanningTask : _10_Drives;
    PROGRAM VisuElems.Visu_Prg WITH VISU_TASK : VisuElems.Visu_Prg;
    PROGRAM _30_Visu WITH VISU_TASK : _30_Visu;
    PROGRAM _40_Vision WITH VisionTask : _40_Vision;
  END_RESOURCE
END_CONFIGURATION

CONFIGURATION SoftMotion General Axis Pool
END_CONFIGURATION

CONFIGURATION SM_Drive_PosControl_J1
END_CONFIGURATION

CONFIGURATION SM_Drive_PosControl_J2
END_CONFIGURATION

CONFIGURATION SM_Drive_PosControl_J3
END_CONFIGURATION

CONFIGURATION SM_Drive_PosControl_J4
END_CONFIGURATION

CONFIGURATION SM_Drive_PosControl_J5
END_CONFIGURATION

CONFIGURATION SM_Drive_PosControl_J6
END_CONFIGURATION

CONFIGURATION <Empty>
END_CONFIGURATION

CONFIGURATION Onewire
END_CONFIGURATION

CONFIGURATION Camera device
END_CONFIGURATION

CONFIGURATION <Empty>
END_CONFIGURATION

CONFIGURATION SPI
END_CONFIGURATION

CONFIGURATION I²C
END_CONFIGURATION

CONFIGURATION I2C_master
END_CONFIGURATION

CONFIGURATION I2C_master_1
END_CONFIGURATION

CONFIGURATION Adafruit_PWM
END_CONFIGURATION

CONFIGURATION AdafruitPwm01
END_CONFIGURATION

CONFIGURATION AdafruitPwm02
END_CONFIGURATION
